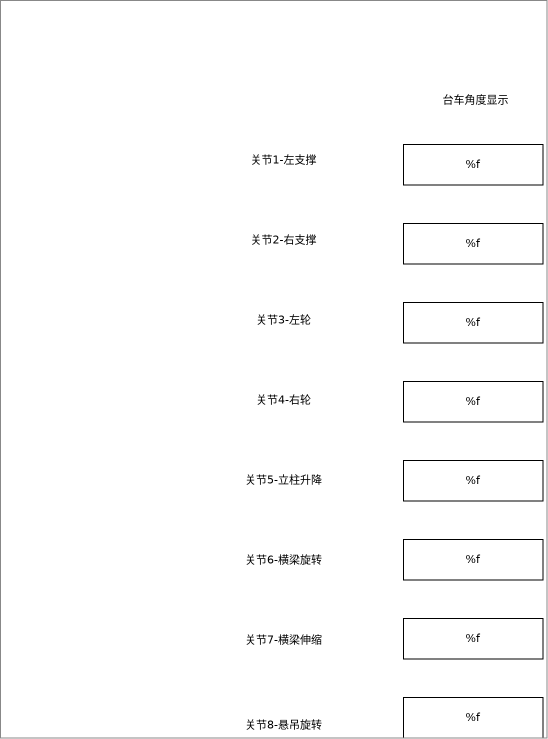
VISUALIZATION motRangeCar  // 548x739
    Label (403,86 145x28), "台车角度显示"
    Label (211,146 145x28), "关节1-左支撑"
    Label (211,226 145x28), "关节2-右支撑"
    Label (211,306 145x28), "关节3-左轮"
    Label (211,386 145x28), "关节4-右轮"
    Label (211,466 145x28), "关节5-立柱升降"
    Label (211,546 145x28), "关节6-横梁旋转"
    Label (211,626 145x28), "关节7-横梁伸缩"
    Label (211,711 145x28), "关节8-悬吊旋转"
    Rectangle (403,144 140x41), "%f", text variable: g_systemInfo.m_cartInfo.m_curJntPosDegMM[1]
    Rectangle (403,223 140x41), "%f", text variable: g_systemInfo.m_cartInfo.m_curJntPosDegMM[2]
    Rectangle (403,302 140x41), "%f", text variable: g_systemInfo.m_cartInfo.m_curJntPosDegMM[3]
    Rectangle (403,381 140x41), "%f", text variable: g_systemInfo.m_cartInfo.m_curJntPosDegMM[4]
    Rectangle (403,460 140x41), "%f", text variable: g_systemInfo.m_cartInfo.m_curJntPosDegMM[5]
    Rectangle (403,539 140x41), "%f", text variable: g_systemInfo.m_cartInfo.m_curJntPosDegMM[6]
    Rectangle (403,618 140x41), "%f", text variable: g_systemInfo.m_cartInfo.m_curJntPosDegMM[7]
    Rectangle (403,697 140x41), "%f", text variable: g_systemInfo.m_cartInfo.m_curJntPosDegMM[8]
END_VISUALIZATION

(* stored: Version 1.1.0.1, ProductVersion 3.1.4024.11
   Visu motRangeCar: Id {b7fecb6d-4394-49ac-8e05-b25fab64cd46} *)
